FUNCTION_BLOCK FB_StackerCrane_Analog
VAR_INPUT
	StackerCraneCurrentPositionXAxis	:	WORD;
	StackerCraneCurrentPositionZAxis	:	WORD;
	ActorInstanceIndex	:	INT;	//Index in DropDown HMI
	ActorInstanceName	:	STRING;		//Name of the instance
END_VAR
VAR_OUTPUT
	SetPointToXAxis : WORD;
	SetPointToZAxis : WORD;
	MoveForkLeft	:	BOOL;
	MoveForkRight	:	BOOL;
END_VAR
VAR_IN_OUT
	OperatingMode	:	OperatingMode;	//Schnittstelle für Betriebsarten
	HMIInterface	:	MachineSectionHMIInterface;	//HMI-Interface
END_VAR
VAR
	statMoveStackerCrane	:	BOOL;
	statStackerCraneInPositionXAxis	:	BOOL;
	statStackerCraneInPositionZAxis	:	BOOL;
	statMoveForkLeft	:	BOOL;
	statMoveForkRight	:	BOOL;
	statCurrentPositionXAxis	: REAL;
	statCurrentPositionZAxis	: REAL;
	statSelectedSetPointXAxis	: REAL;
	statSelectedSetPointZAxis	: REAL;
	statSetPointXAxis	:	REAL;
	statSetPointZAxis	:	REAL;
	statSetPointToXaxis	:	WORD;
	statSetPointToZaxis	:	WORD;
	
	internHMIInterface	:	MachineSectionHMIInterface;
	internInstanceActivatedFirstTime	:	BOOL;
	internRisingEdgePressButtonUpXAxis	:	R_TRIG;
	internRisingEdgePressButtonDownXAxis	:	R_TRIG;
	internRisingEdgePressButtonStopXAxis	:	R_TRIG;
	internRisingEdgePressButtonUpZAxis	:	R_TRIG;
	internRisingEdgePressButtonDownZAxis	:	R_TRIG;
	internRisingEdgePressButtonStopZAxis	:	R_TRIG;
	internRisingEdgePressButtonForkLeft	:	R_TRIG;
	internRisingEdgePressButtonForkRight	:	R_TRIG;
	internRisingEdgePressButtonMiddleFork	:	R_TRIG;
	internStopXAxis	:	BOOL;
	internStopZAxis	:	BOOL;
	internMiddleFork	:	BOOL;
END_VAR

(*===================== CurrentPosition Axes =====================*)
FC_AnalogInputValueHandling(RowValue:= StackerCraneCurrentPositionXAxis, 
							UpperLimit:= 10.5, 
							LowerLimit:= 0.0, 
							ConvertedValue=> statCurrentPositionXAxis);
FC_AnalogInputValueHandling(RowValue:= StackerCraneCurrentPositionZAxis, 
							UpperLimit:= 6.625, 
							LowerLimit:= 0.0, 
							ConvertedValue=> statCurrentPositionZAxis);
(*===================== HMI INTERFACE =====================*)
internHMIInterface := HMIInterface;

IF internHMIInterface.ActiveMachineSection = MachineSection.StackerCrane AND
	internHMIInterface.SelectedActor = ActorInstanceIndex THEN
	(*===================== Initializing HMI-Interface =====================*)
	IF NOT internInstanceActivatedFirstTime THEN
		FC_InitializingSettingLines(HMIInterface := internHMIInterface);
		internInstanceActivatedFirstTime := TRUE;
	END_IF
	(*===================== Button Handling Movement =====================*)
	internHMIInterface.Movements.MovementSettingLines[1].CaptionSettingLine := CONCAT('StackerCrane X-Axis Control ', ActorInstanceName);
	internHMIInterface.Movements.MovementSettingLines[1].VisibilitySettingLine := TRUE;
	
	internHMIInterface.Movements.MovementSettingLines[1].SettingLineButtons[1].IsVisibleButton := TRUE;
	internHMIInterface.Movements.MovementSettingLines[1].SettingLineButtons[1].IsVisibleAxisPosition := FALSE;
	internHMIInterface.Movements.MovementSettingLines[1].SettingLineButtons[1].IsEnabled := OperatingMode.ManuelIsActive AND NOT
									 														OperatingMode.EStop.IsActive AND NOT
																							OperatingMode.Fault.IsActive AND NOT
																							statMoveStackerCrane AND
																							statSetPointXAxis < 10.5;
	internHMIInterface.Movements.MovementSettingLines[1].SettingLineButtons[1].InPosition := statStackerCraneInPositionXAxis;
	internHMIInterface.Movements.MovementSettingLines[1].SettingLineButtons[1].CaptionButton := 'Right';
	internHMIInterface.Movements.MovementSettingLines[1].SettingLineButtons[1].PathImageButton := 'Images\ForwardConveyor.svg';
	
	internHMIInterface.Movements.MovementSettingLines[1].SettingLineButtons[2].IsVisibleButton := TRUE;
	internHMIInterface.Movements.MovementSettingLines[1].SettingLineButtons[2].IsVisibleAxisPosition := TRUE;
	internHMIInterface.Movements.MovementSettingLines[1].SettingLineButtons[2].IsEnabled := OperatingMode.ManuelIsActive;
	internHMIInterface.Movements.MovementSettingLines[1].SettingLineButtons[2].InPosition := NOT statMoveStackerCrane;
	internHMIInterface.Movements.MovementSettingLines[1].SettingLineButtons[2].AxisPosition := statCurrentPositionXAxis;
	internHMIInterface.Movements.MovementSettingLines[1].SettingLineButtons[2].CaptionButton := 'Stop';
	internHMIInterface.Movements.MovementSettingLines[1].SettingLineButtons[2].PathImageButton := 'Images\StopConveyor.svg';
	
	internHMIInterface.Movements.MovementSettingLines[1].SettingLineButtons[3].IsVisibleButton := TRUE;
	internHMIInterface.Movements.MovementSettingLines[1].SettingLineButtons[3].IsVisibleAxisPosition := FALSE;
	internHMIInterface.Movements.MovementSettingLines[1].SettingLineButtons[3].IsEnabled := OperatingMode.ManuelIsActive AND NOT
									 														OperatingMode.EStop.IsActive AND NOT
																							OperatingMode.Fault.IsActive AND NOT
																							statMoveStackerCrane AND
																							statSetPointXAxis > 0;
	internHMIInterface.Movements.MovementSettingLines[1].SettingLineButtons[3].InPosition := statStackerCraneInPositionXAxis;
	internHMIInterface.Movements.MovementSettingLines[1].SettingLineButtons[3].CaptionButton := 'Left';
	internHMIInterface.Movements.MovementSettingLines[1].SettingLineButtons[3].PathImageButton := 'Images\BackwardConveyor.svg';
	
	internHMIInterface.Movements.MovementSettingLines[2].CaptionSettingLine := CONCAT('StackerCrane Z-Axis Control ', ActorInstanceName);
	internHMIInterface.Movements.MovementSettingLines[2].VisibilitySettingLine := TRUE;
	
	internHMIInterface.Movements.MovementSettingLines[2].SettingLineButtons[1].IsVisibleButton := TRUE;
	internHMIInterface.Movements.MovementSettingLines[2].SettingLineButtons[1].IsVisibleAxisPosition := FALSE;
	internHMIInterface.Movements.MovementSettingLines[2].SettingLineButtons[1].IsEnabled := OperatingMode.ManuelIsActive AND NOT
									 														OperatingMode.EStop.IsActive AND NOT
																							OperatingMode.Fault.IsActive AND NOT
																							statMoveStackerCrane AND
																							statSetPointZAxis < 10.5;
	internHMIInterface.Movements.MovementSettingLines[2].SettingLineButtons[1].InPosition := statStackerCraneInPositionZAxis;
	internHMIInterface.Movements.MovementSettingLines[2].SettingLineButtons[1].CaptionButton := 'Up';
	internHMIInterface.Movements.MovementSettingLines[2].SettingLineButtons[1].PathImageButton := 'Images\UpElevator.svg';
	
	internHMIInterface.Movements.MovementSettingLines[2].SettingLineButtons[2].IsVisibleButton := TRUE;
	internHMIInterface.Movements.MovementSettingLines[2].SettingLineButtons[2].IsVisibleAxisPosition := TRUE;
	internHMIInterface.Movements.MovementSettingLines[2].SettingLineButtons[2].IsEnabled := OperatingMode.ManuelIsActive;
	internHMIInterface.Movements.MovementSettingLines[2].SettingLineButtons[2].InPosition := NOT statMoveStackerCrane;
	internHMIInterface.Movements.MovementSettingLines[2].SettingLineButtons[2].AxisPosition := statCurrentPositionZAxis;
	internHMIInterface.Movements.MovementSettingLines[2].SettingLineButtons[2].CaptionButton := 'Stop';
	internHMIInterface.Movements.MovementSettingLines[2].SettingLineButtons[2].PathImageButton := 'Images\StopConveyor.svg';
	
	internHMIInterface.Movements.MovementSettingLines[2].SettingLineButtons[3].IsVisibleButton := TRUE;
	internHMIInterface.Movements.MovementSettingLines[2].SettingLineButtons[3].IsVisibleAxisPosition := FALSE;
	internHMIInterface.Movements.MovementSettingLines[2].SettingLineButtons[3].IsEnabled := OperatingMode.ManuelIsActive AND NOT
									 														OperatingMode.EStop.IsActive AND NOT
																							OperatingMode.Fault.IsActive AND NOT
																							statMoveStackerCrane AND
																							statSetPointZAxis > 0;
	internHMIInterface.Movements.MovementSettingLines[2].SettingLineButtons[3].InPosition := statStackerCraneInPositionXAxis;
	internHMIInterface.Movements.MovementSettingLines[2].SettingLineButtons[3].CaptionButton := 'Down';
	internHMIInterface.Movements.MovementSettingLines[2].SettingLineButtons[3].PathImageButton := 'Images\DownElevator.svg';
	
	internHMIInterface.Forks.ForkMovementSettingLines[1].CaptionSettingLine := CONCAT('Fork Control ', ActorInstanceName);
	internHMIInterface.Forks.ForkMovementSettingLines[1].VisibilitySettingLine := TRUE;
	
	internHMIInterface.Forks.ForkMovementSettingLines[1].SettingLineButtons[1].IsVisibleButton := TRUE;
	internHMIInterface.Forks.ForkMovementSettingLines[1].SettingLineButtons[1].IsVisibleAxisPosition := FALSE;
	internHMIInterface.Forks.ForkMovementSettingLines[1].SettingLineButtons[1].IsEnabled := OperatingMode.ManuelIsActive AND NOT
									 														OperatingMode.EStop.IsActive AND NOT
																							OperatingMode.Fault.IsActive AND NOT
																							statMoveStackerCrane AND
																							statStackerCraneInPositionXAxis AND
																							statStackerCraneInPositionZAxis;
	internHMIInterface.Forks.ForkMovementSettingLines[1].SettingLineButtons[1].InPosition := statMoveForkLeft;
	internHMIInterface.Forks.ForkMovementSettingLines[1].SettingLineButtons[1].CaptionButton := 'Left';
	internHMIInterface.Forks.ForkMovementSettingLines[1].SettingLineButtons[1].PathImageButton := 'Images\BackwardConveyor.svg';
	
	internHMIInterface.Forks.ForkMovementSettingLines[1].SettingLineButtons[2].IsVisibleButton := TRUE;
	internHMIInterface.Forks.ForkMovementSettingLines[1].SettingLineButtons[2].IsVisibleAxisPosition := FALSE;
	internHMIInterface.Forks.ForkMovementSettingLines[1].SettingLineButtons[2].IsEnabled := OperatingMode.ManuelIsActive;
	internHMIInterface.Forks.ForkMovementSettingLines[1].SettingLineButtons[2].InPosition := NOT statMoveForkLeft AND NOT statMoveForkRight;
	internHMIInterface.Forks.ForkMovementSettingLines[1].SettingLineButtons[2].CaptionButton := 'Stop';
	internHMIInterface.Forks.ForkMovementSettingLines[1].SettingLineButtons[2].PathImageButton := 'Images\StopConveyor.svg';
	
	internHMIInterface.Forks.ForkMovementSettingLines[1].SettingLineButtons[3].IsVisibleButton := TRUE;
	internHMIInterface.Forks.ForkMovementSettingLines[1].SettingLineButtons[3].IsVisibleAxisPosition := FALSE;
	internHMIInterface.Forks.ForkMovementSettingLines[1].SettingLineButtons[3].IsEnabled := OperatingMode.ManuelIsActive AND NOT
									 														OperatingMode.EStop.IsActive AND NOT
																							OperatingMode.Fault.IsActive AND NOT
																							statMoveStackerCrane AND
																							statStackerCraneInPositionXAxis AND
																							statStackerCraneInPositionZAxis;
	internHMIInterface.Forks.ForkMovementSettingLines[1].SettingLineButtons[3].InPosition := statMoveForkRight;
	internHMIInterface.Forks.ForkMovementSettingLines[1].SettingLineButtons[3].CaptionButton := 'Right';
	internHMIInterface.Forks.ForkMovementSettingLines[1].SettingLineButtons[3].PathImageButton := 'Images\ForwardConveyor.svg';
	
	(*===================== X-Axis Up =====================*)
	internRisingEdgePressButtonUpXAxis(CLK := internHMIInterface.Movements.MovementSettingLines[1].SettingLineButtons[1].IsPressed);
	IF internRisingEdgePressButtonUpXAxis.Q THEN
		statSetPointXAxis := statSetPointXAxis + 0.2;
		statMoveStackerCrane := TRUE;
	END_IF
	(*===================== X-Axis Down =====================*)
	internRisingEdgePressButtonDownXAxis(CLK := internHMIInterface.Movements.MovementSettingLines[1].SettingLineButtons[3].IsPressed);
	IF internRisingEdgePressButtonDownXAxis.Q THEN
		statSetPointXAxis := statSetPointXAxis - 0.2;
		statMoveStackerCrane := TRUE;
	END_IF
	(*===================== X-Axis Stop =====================*)
	internRisingEdgePressButtonStopXAxis(CLK := internHMIInterface.Movements.MovementSettingLines[1].SettingLineButtons[2].IsPressed);
	IF internRisingEdgePressButtonStopXAxis.Q THEN
		internStopXAxis := TRUE;
	END_IF
	(*===================== Z-Axis Up =====================*)
	internRisingEdgePressButtonUpZAxis(CLK := internHMIInterface.Movements.MovementSettingLines[2].SettingLineButtons[1].IsPressed);
	IF internRisingEdgePressButtonUpZAxis.Q THEN
		statSetPointZAxis := statSetPointZAxis + 0.2;
		statMoveStackerCrane := TRUE;
	END_IF
	(*===================== Z-Axis Down =====================*)
	internRisingEdgePressButtonDownZAxis(CLK := internHMIInterface.Movements.MovementSettingLines[2].SettingLineButtons[3].IsPressed);
	IF internRisingEdgePressButtonDownZAxis.Q THEN
		statSetPointZAxis := statSetPointZAxis - 0.2;
		statMoveStackerCrane := TRUE;
	END_IF
	(*===================== Z-Axis Stop =====================*)
	internRisingEdgePressButtonStopZAxis(CLK := internHMIInterface.Movements.MovementSettingLines[2].SettingLineButtons[2].IsPressed);
	IF internRisingEdgePressButtonStopZAxis.Q THEN
		internStopZAxis := TRUE;
	END_IF
	(*===================== Fork Left =====================*)
	internRisingEdgePressButtonForkLeft(CLK := internHMIInterface.Forks.ForkMovementSettingLines[1].SettingLineButtons[1].IsPressed);
	IF internRisingEdgePressButtonForkLeft.Q THEN
		statMoveForkLeft := TRUE;
	END_IF
	(*===================== Fork Right =====================*)
	internRisingEdgePressButtonForkRight(CLK := internHMIInterface.Forks.ForkMovementSettingLines[1].SettingLineButtons[3].IsPressed);
	IF internRisingEdgePressButtonForkRight.Q THEN
		statMoveForkRight := TRUE;
	END_IF
	(*===================== Fork Middle =====================*)
	internRisingEdgePressButtonMiddleFork(CLK := internHMIInterface.Forks.ForkMovementSettingLines[1].SettingLineButtons[2].IsPressed);
	IF internRisingEdgePressButtonMiddleFork.Q THEN
		statMoveForkLeft := FALSE;
		statMoveForkRight := FALSE;
	END_IF
	
	(*===================== Write Interface =====================*)
	HMIInterface := internHMIInterface;
ELSE
		internInstanceActivatedFirstTime := FALSE;
END_IF
(*===================== Stacker crane in Position =====================*)
EvaluatePosition();
(*===================== Positioning Stacker crane =====================*)
IF ((OperatingMode.AutomaticIsActive AND OperatingMode.AutomaticStart.IsActive) OR
	(OperatingMode.ManuelIsActive)) 
   AND statMoveStackerCrane 
THEN
	statSelectedSetPointXAxis := statSetPointXAxis;
	statSelectedSetPointZAxis := statSetPointZAxis;
END_IF
IF OperatingMode.EStop.IsActive OR OperatingMode.Fault.IsActive OR 
((OperatingMode.AutomaticIsActive AND OperatingMode.AutomaticStop.IsActive) OR
(OperatingMode.ManuelIsActive AND (internStopXAxis OR internStopZAxis)))
THEN
	statSelectedSetPointXAxis := statCurrentPositionXAxis;
	statSelectedSetPointZAxis := statCurrentPositionZAxis;
	statMoveStackerCrane := FALSE;
END_IF
(*===================== SetPoint X-Axis =====================*)
FC_AnalogOutputValueHandling(Setpoint:= statSelectedSetPointXAxis, 
						     UpperLimit:= 10.5, 
							 LowerLimit:= 0.0, 
							 ConvertedValue=> statSetPointToXaxis);
(*===================== SetPoint Z-Axis =====================*)
FC_AnalogOutputValueHandling(Setpoint:= statSelectedSetPointZAxis, 
						     UpperLimit:= 6.625, 
							 LowerLimit:= 0.0, 
							 ConvertedValue=> statSetPointToZaxis);
(*===================== Outputs writting =====================*)
SetPointToXAxis := statSetPointToXaxis;
SetPointToZAxis := statSetPointToZaxis;
MoveForkLeft := statMoveForkLeft;
MoveForkRight := statMoveForkRight;

METHOD PUBLIC EvaluatePosition
IF statStackerCraneInPositionXAxis AND statStackerCraneInPositionZAxis THEN
	statMoveStackerCrane := FALSE;
END_IF
IF (statCurrentPositionXAxis >= statSetPointXAxis - 0.1) AND (statCurrentPositionXAxis <= statSetPointXAxis + 0.1) THEN
	statStackerCraneInPositionXAxis := TRUE;
ELSE
	statStackerCraneInPositionXAxis := FALSE;
END_IF
IF (statCurrentPositionZAxis >= statSetPointZAxis - 0.1) AND (statCurrentPositionZAxis <= statSetPointZAxis + 0.1) THEN
	statStackerCraneInPositionZAxis := TRUE;
ELSE
	statStackerCraneInPositionZAxis := FALSE;
END_IF
END_METHOD

PROPERTY PUBLIC InPositionXAxis : BOOL
GET
InPositionXAxis := statStackerCraneInPositionXAxis;
END_GET
END_PROPERTY

PROPERTY PUBLIC InPositionZAxis : BOOL
GET
InPositionZAxis := statStackerCraneInPositionZAxis;
END_GET
END_PROPERTY

METHOD PUBLIC MoveAxesStackerCrane_ON : BOOL
VAR_INPUT
	StartMoveStackerCrane	:	BOOL;
	PositionXAxis	:	REAL;
	PositionZAxis	:	REAL;
END_VAR
IF OperatingMode.AutomaticIsActive AND OperatingMode.AutomaticStart.IsActive AND
	NOT statMoveStackerCrane AND StartMoveStackerCrane THEN
	SetPointXAxis := PositionXAxis;
	SetPointZAxis := PositionZAxis;
	statMoveStackerCrane := TRUE;
// 	statStackerCraneInPositionXAxis := FALSE;
// 	statStackerCraneInPositionZAxis := FALSE;
END_IF
END_METHOD

METHOD PUBLIC MoveForkToLeft_ON : BOOL
VAR_INPUT
	StartMovingForkLeft	:	BOOL;
END_VAR
IF OperatingMode.AutomaticIsActive AND OperatingMode.AutomaticStart.IsActive AND
	InPositionXAxis AND InPositionZAxis AND StartMovingForkLeft AND NOT statMoveStackerCrane 
THEN
	statMoveForkLeft := TRUE;
	MoveForkToLeft_ON := TRUE;
ELSE
	MoveForkToLeft_ON := FALSE;
END_IF
END_METHOD

METHOD PUBLIC MoveForkToMiddle_ON : BOOL
VAR_INPUT
	StartMovingForkMiddle: BOOL;
END_VAR
IF OperatingMode.AutomaticIsActive AND OperatingMode.AutomaticStart.IsActive AND 
	StartMovingForkMiddle THEN
	statMoveForkLeft := FALSE;
	statMoveForkRight := FALSE;
	MoveForkToMiddle_ON := TRUE;
ELSE
	MoveForkToMiddle_ON := FALSE;
END_IF
END_METHOD

METHOD PUBLIC MoveForkToRight_ON : BOOL
VAR_INPUT
	StartMovingForkRight	:	BOOL;
END_VAR
IF OperatingMode.AutomaticIsActive AND OperatingMode.AutomaticStart.IsActive AND
	InPositionXAxis AND InPositionZAxis AND StartMovingForkRight  AND NOT statMoveStackerCrane
THEN
	statMoveForkRight := TRUE;
	MoveForkToRight_ON := TRUE;
ELSE
	MoveForkToRight_ON := FALSE;
END_IF
END_METHOD

PROPERTY PUBLIC SetPointXAxis : REAL
GET
SetPointXAxis := statSetPointXAxis;
END_GET
SET
IF SetPointXAxis < 10.5 THEN
	statSetPointXAxis := SetPointXAxis;
END_IF
END_SET
END_PROPERTY

PROPERTY PUBLIC SetPointZAxis : REAL
GET
SetPointZAxis := statSetPointZAxis;
END_GET
SET
IF SetPointZAxis < 6.125 THEN
	statSetPointZAxis := SetPointZAxis;	
END_IF
END_SET
END_PROPERTY

END_FUNCTION_BLOCK

(* stored: Version 1.1.0.1
   POU FB_StackerCrane_Analog: Id {b4e2a7dd-fd58-4b61-a413-e8e9cbb651c1}, SpecialFunc None
   Method EvaluatePosition: Id {009b1d40-db45-4d5b-9724-104d00ffa9de}
   Property InPositionXAxis: Id {99b77603-dec4-46a3-af14-48acaf9c0f42}
   Get Get: Id {b62af317-8d1c-4248-aa9c-84fbfdf53b86}
   Property InPositionZAxis: Id {a0b014ec-cf84-488b-a248-e9ae88e49c90}
   Get Get: Id {451cccd6-9c41-495b-bdf1-e7527ebb369a}
   Method MoveAxesStackerCrane_ON: Id {8267f457-7374-46a9-a364-11d0c21ace83}
   Method MoveForkToLeft_ON: Id {e5457c5c-a9f1-4c16-a39b-9e4696966196}
   Method MoveForkToMiddle_ON: Id {6c553420-83ab-4b81-b720-d2d4660e261f}
   Method MoveForkToRight_ON: Id {f02a451c-62d7-4e7b-bbbb-17a3b3d967b4}
   Property SetPointXAxis: Id {7280cb07-7183-4572-9de9-19d1fca068b7}
   Get Get: Id {d62e30d2-cf9a-4efb-b797-b8a90938b1b9}
   Set Set: Id {7a08d128-5616-425e-8ec6-156b19d1eb78}
   Property SetPointZAxis: Id {d7138e03-dbd8-465a-8b2a-1e9badd135cc}
   Get Get: Id {bb04fd2d-5cab-4cda-848d-1d129d9416ea}
   Set Set: Id {f49d28a9-7efb-4e8a-bdae-3981713b245d} *)
